(* This function block is created for interface devices between different PLC*)
(* Not all the fields in the original structure is required, just few signals *)
(*Use with FB_ADS_WATCHDOG on remotePLC*)
FUNCTION_BLOCK FB_TVGC_2S_ADS extends FB_ADS
VAR_INPUT
    sNetId : String; //NetID of the Destination PLC controller
    nPort : UINT; // port number
    sVarName : string;// the variable name of the (device) declared function block.
    iWatchdog:UDINT;//The watchdog variable name written to by the remote plc
END_VAR
VAR_OUTPUT
    {attribute 'pytmc' := 'pv: '}
    VGC:ST_VGC_2S;
    bError:BOOL;
END_VAR
VAR
    fb_CheckWatchdog: FB_CheckWatchdog;
    fb_Read_VGC: FB_ReadAdsSymByName;
    ftReset: F_TRIG;
    xFirstPass: bool:= true;
END_VAR

ftReset(CLK:= fb_Read_VGC.bBusy OR xFirstPass);
xFirstPass:=false;
(*calling ADS read function*)
fb_Read_VGC(
    bRead:= ftReset.Q,
    sNetId:= sNetId,
    nPort:= nPort,
    sVarName:= CONCAT(sVarName,'.iq_stValve'),
    nDestAddr:= ADR(VGC),
    nLen:= SIZEOF(VGC),
    tTimeout:= ,
    eComMode:= eAdsComModeFastCom,
    bBusy=> ,
    bError=> ,
    nErrorId=> );


(*Error*)
fb_CheckWatchdog(
    bEnable:= TRUE,
    tWatchdogTime:= T#900ms,
    nCnt:= iWatchdog ,
    bWatchdog=> ,
    nLastCnt=> );
bError:= fb_Read_VGC.bError OR fb_CheckWatchdog.bWatchdog;

ACT_Logger();

ACTION ACT_Logger:
IF tErrorPresent.Q THEN
 IF(fb_Read_VGC.bError) THEN fbLogger(sMsg:='ADS Read Error', eSevr:=TcEventSeverity.Critical); END_IF;
 IF(fb_CheckWatchdog.bWatchdog) THEN fbLogger(sMsg:='ADS Watchdog Error', eSevr:=TcEventSeverity.Critical); END_IF;
END_IF
END_ACTION

END_FUNCTION_BLOCK

(* stored: Version 1.1.0.1
   POU FB_TVGC_2S_ADS: Id {2d33fb71-254e-4ee8-8b31-f9715402f769}, SpecialFunc None
   Action ACT_Logger: Id {4dcca01b-a24b-4b1b-865e-ad4d9c835d32} *)
